FUNCTION TryConvert_REAL_TO_LWORD : BOOL
VAR_INPUT
	in : REAL;
	out : REFERENCE TO LWORD;
END_VAR

IF in > DatatypeLimits.MAX_VALUE_OF_REAL_WHICH_CAN_BE_HELD_IN_A_LWORD THEN
	RETURN;
END_IF

IF in < DatatypeLimits.MIN_VALUE_OF_REAL_WHICH_CAN_BE_HELD_IN_A_LWORD THEN
	RETURN;
END_IF

out := REAL_TO_LWORD(in);
TryConvert_REAL_TO_LWORD := TRUE;

END_FUNCTION

(* stored: Version 1.1.0.1, ProductVersion 3.1.4024.12
   POU TryConvert_REAL_TO_LWORD: Id {4a64edbe-f2d7-4097-baa6-597450838768}, SpecialFunc None *)
